// TIA Portal V18 export
// export: Created 2026-06-08T17:01:57.992056Z, ExportSetting WithDefaults, DisplayName Totally Integrated Automation Portal, DisplayVersion V18, DisplayName TIA Portal Openness, DisplayVersion V18, DisplayName TIA Portal Version Control Interface, DisplayVersion V18, DisplayName STEP 7 Professional, DisplayVersion V18, DisplayName STEP 7 Safety, DisplayVersion V18, DisplayName WinCC Professional, DisplayVersion V18
FUNCTION "MAIN_I/O" : Void   // FC1, LAD
{ S7_Optimized_Access := 'TRUE' }
VERSION : 0.1
// stored: AutoNumber true, IsIECCheckEnabled false, SetENOAutomatically false, UDAEnableTagReadback false
BEGIN

REGION Network 1
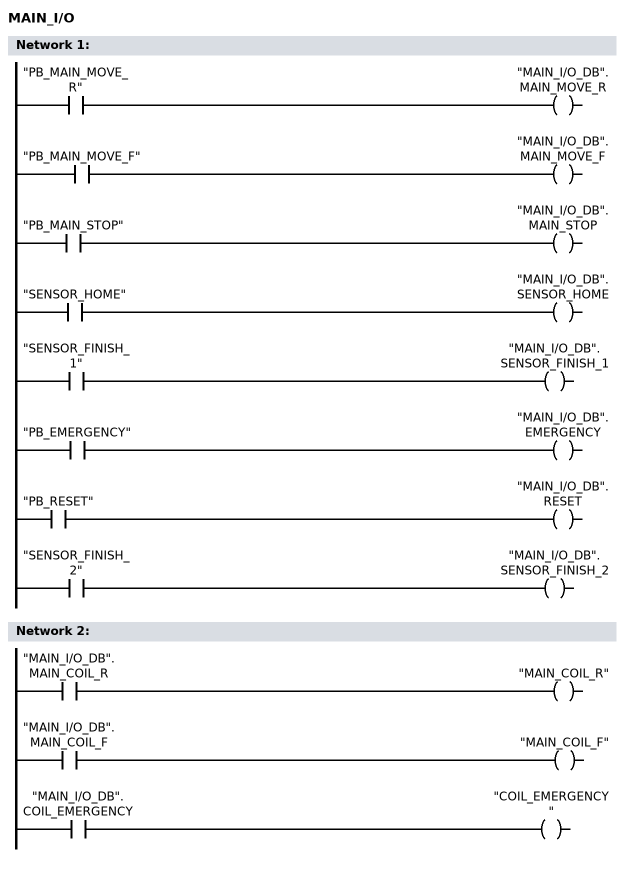
   RUNG wire#powerrail
      Contact( "PB_MAIN_MOVE_R" )
      Coil( "MAIN_I/O_DB".MAIN_MOVE_R )
   END_RUNG
   RUNG wire#powerrail
      Contact( "PB_MAIN_MOVE_F" )
      Coil( "MAIN_I/O_DB".MAIN_MOVE_F )
   END_RUNG
   RUNG wire#powerrail
      Contact( "PB_MAIN_STOP" )
      Coil( "MAIN_I/O_DB".MAIN_STOP )
   END_RUNG
   RUNG wire#powerrail
      Contact( "SENSOR_HOME" )
      Coil( "MAIN_I/O_DB".SENSOR_HOME )
   END_RUNG
   RUNG wire#powerrail
      Contact( "SENSOR_FINISH_1" )
      Coil( "MAIN_I/O_DB".SENSOR_FINISH_1 )
   END_RUNG
   RUNG wire#powerrail
      Contact( "PB_EMERGENCY" )
      Coil( "MAIN_I/O_DB".EMERGENCY )
   END_RUNG
   RUNG wire#powerrail
      Contact( "PB_RESET" )
      Coil( "MAIN_I/O_DB".RESET )
   END_RUNG
   RUNG wire#powerrail
      Contact( "SENSOR_FINISH_2" )
      Coil( "MAIN_I/O_DB".SENSOR_FINISH_2 )
   END_RUNG
   // the same network as SCL:
   "MAIN_I/O_DB".MAIN_MOVE_R := "PB_MAIN_MOVE_R";
   "MAIN_I/O_DB".MAIN_MOVE_F := "PB_MAIN_MOVE_F";
   "MAIN_I/O_DB".MAIN_STOP := "PB_MAIN_STOP";
   "MAIN_I/O_DB".SENSOR_HOME := "SENSOR_HOME";
   "MAIN_I/O_DB".SENSOR_FINISH_1 := "SENSOR_FINISH_1";
   "MAIN_I/O_DB".EMERGENCY := "PB_EMERGENCY";
   "MAIN_I/O_DB".RESET := "PB_RESET";
   "MAIN_I/O_DB".SENSOR_FINISH_2 := "SENSOR_FINISH_2";
END_REGION

REGION Network 2
   RUNG wire#powerrail
      Contact( "MAIN_I/O_DB".MAIN_COIL_R )
      Coil( "MAIN_COIL_R" )
   END_RUNG
   RUNG wire#powerrail
      Contact( "MAIN_I/O_DB".MAIN_COIL_F )
      Coil( "MAIN_COIL_F" )
   END_RUNG
   RUNG wire#powerrail
      Contact( "MAIN_I/O_DB".COIL_EMERGENCY )
      Coil( "COIL_EMERGENCY" )
   END_RUNG
   // the same network as SCL:
   "MAIN_COIL_R" := "MAIN_I/O_DB".MAIN_COIL_R;
   "MAIN_COIL_F" := "MAIN_I/O_DB".MAIN_COIL_F;
   "COIL_EMERGENCY" := "MAIN_I/O_DB".COIL_EMERGENCY;
END_REGION
END_FUNCTION
